TYPE stPose2D EXTENDS stPose :
STRUCT
	theta : LREAL;
END_STRUCT
END_TYPE

(* stored: Version 1.1.0.1, ProductVersion 3.1.4026.18
   DUT stPose2D: Id {b1b2c3d4-4444-4444-4444-444444444444} *)
